TYPE "udt_LinTranformation"
VERSION : 0.1
// Block: udt_LinTranformation
   STRUCT
      m : Real;
      q : Real;
   END_STRUCT;

END_TYPE
